# EPICS autosave request: eurotherm2k/eurotherm2k_settings.req
$(P)$(Q):PID.SCAN
$(P)$(Q):UPDATE.SCAN
